// TIA Portal V19 export
TYPE "PPrf_Rollformer"
// stored: Access Published
   STRUCT
      Code : UInt;
      FAK : LReal;
      Acc : LReal;
      Dec : LReal;
      Jerk : LReal;
      TAxConfig : Struct
         EncoderInverseDirection : Bool;
         MotorInverseDirection : Bool;
         LoadGearNumerator : UDInt;
         LoadGearDenominator : UDInt;
         MechanicsLeadScrew : LReal;
         EncoderDistancePerRevolution : LReal;
         DynamicsLimitsMaxVelocity : LReal;   // Dynamic limitation for maximum speed (mechanical)
         DynamicsLimitsVelocity : LReal;   // Dynamic limitation for maximum speed (programmable)
         ControlLoop_Kv : LReal;   // <TO>.PositionControl.Kv
         ControlLoop_Kpc : LReal;   // <TO>.PositionControl.Kpc
         ControlLoop_Vtc : LReal;   // <TO>.DynamicAxisModel.VelocityTimeConstant
      END_STRUCT;
   END_STRUCT;
END_TYPE
